TYPE XMLHeader :
STRUCT
	MaschineNummer : STRING:= '1234567890';
	Manufacturer : STRING := 'Beckhoff';
	Maschinetype : STRING:= 'cx2040.1.1.1';
	Customer : STRING:= 'liyizhen23333';
END_STRUCT
END_TYPE

(* stored: Version 1.1.0.1, ProductVersion 3.1.4024.3
   DUT XMLHeader: Id {04aaf20d-1a56-4173-999c-2a06f76d84aa} *)
